// Motor with one direction
FUNCTION_BLOCK FB_Motor
VAR_INPUT
	bAlarmSignal: BOOL;        // NC alarm signal from the device
END_VAR
VAR_OUTPUT
	bRun: BOOL;                // Output to run the motor
	bError: BOOL;              // Motor is in error
END_VAR
VAR
END_VAR

IF inError THEN                // Stop the motor if it is in th error state
	Stop();
	bError := TRUE;
ELSE
	bError := FALSE;
END_IF

// Motor is in the error state
PROPERTY inError : Bool
GET
inError := NOT bAlarmSignal;
END_GET
END_PROPERTY

PROPERTY isStoped : Bool
GET
IsStoped := (bRun = FALSE);
END_GET
END_PROPERTY

// Run the motor
METHOD Run : BOOL
VAR_INPUT
END_VAR
bRun := TRUE; // Set output for motor to run
END_METHOD

// Stop the motor
METHOD Stop : BOOL
VAR_INPUT
END_VAR
bRun := FALSE; // Reset output for motor to run
END_METHOD

END_FUNCTION_BLOCK

(* stored: Version 1.1.0.1, ProductVersion 3.1.4024.12
   POU FB_Motor: Id {f3102ce1-fae7-4431-8264-728e8d939b92}, SpecialFunc None
   Property inError: Id {3d652894-fd98-4a1d-8e97-37f9219b5940}
   Get Get: Id {f0058e0e-7c3c-401d-b2c5-47887384743d}
   Property isStoped: Id {b6975c72-b2db-4f16-ae75-d5ea8cc68af0}
   Get Get: Id {b09331fe-f9d9-4fc8-99e7-4d367c9dafbd}
   Method Run: Id {eb5d2897-9226-4b06-a6c6-14e8c4b45c46}
   Method Stop: Id {6100c783-cc3d-41b2-86eb-0dcea861185a} *)
